TYPE stMOVIKITpositioningDrive :
STRUCT
	IN: stPositioning_IN;
	OUT: stPositioning_OUT;
	ApplicationMode: eMOVIKITpositioningDrive_ApplMode;
	
END_STRUCT
END_TYPE

(* stored: Version 1.1.0.1, ProductVersion 3.1.4024.9
   DUT stMOVIKITpositioningDrive: Id {1cdb44a8-26fa-46ea-a191-3cc94837c8d3} *)
